// TwinCAT 3 PLC project Untitled1
// ProgramVersion: 3.1.4023.0
// libraries:
//   Tc2_Standard, * (Beckhoff Automation GmbH)
//   Tc2_System, * (Beckhoff Automation GmbH)
//   Tc3_Module, * (Beckhoff Automation GmbH)
//   VisuSymbols,3.5.10.0,System
// project tree:
//   / GlobalTextList.TcGTLO, PlcTask.TcTTO, RecipeManager.TcRMO (not stored), Visualization Manager.TcVMO (not stored), VISU_TASK.TcTTO
//   GVLs/ Recipes.TcGVL
//   POUs/ FB_PIZZA_OVEN.TcPOU, MAIN.TcPOU
//   VISUs/ OvenSimulation.TcVIS

CONFIGURATION Untitled1
    RESOURCE PLC ON TwinCAT3
        TASK PlcTask(INTERVAL := T#10ms, PRIORITY := 20);
        TASK VISU_TASK(INTERVAL := T#200000us, PRIORITY := 30);
        PROGRAM MAIN WITH PlcTask : MAIN;
        PROGRAM VisuElems_Visu_Prg WITH VISU_TASK : VisuElems.Visu_Prg;
    END_RESOURCE
END_CONFIGURATION

// ---- GVLs/Recipes.TcGVL
{attribute 'qualified_only'}
VAR_GLOBAL
END_VAR

// ---- POUs/MAIN.TcPOU
PROGRAM MAIN
VAR

	fbMyPizzaOven:FB_PIZZA_OVEN; //oven 1
	fbMyPizzaOven2:FB_PIZZA_OVEN; //oven 2
	btn_PutAPizza:BOOL;
	btn_PackageThePizza:BOOL;
	bReset:BOOL;
	
	btn_PutAPizzaT:R_TRIG;
	btn_PackageThePizzaT:R_TRIG;
	bResetT:R_TRIG;
	
	fbReadRecipe:RecipeManCommands;
	btnLoadRecipe:BOOL;
	btnSaveRecipe:BOOL;
	iIndexRecipe:int;
END_VAR

btn_PutAPizzaT(CLK:=main.btn_PutAPizza);
btn_PackageThePizzaT(CLK:=main.btn_PackageThePizza);
bResetT(CLK:=main.bReset);

fbMyPizzaOven(
	bReset:=main.bResetT.Q,
	btn_PutAPizza:=main.btn_PutAPizzaT.Q,
	btn_PackageThePizza:=main.btn_PackageThePizzaT.Q
);

fbMyPizzaOven2(
	bReset:=main.bResetT.Q,
	btn_PutAPizza:=main.btn_PutAPizzaT.Q,
	btn_PackageThePizza:=main.btn_PackageThePizzaT.Q
);

IF btnSaveRecipe THEN
	fbReadRecipe.ReadRecipe(
		RecipeDefinitionName:='Recipe',
		RecipeName:='MyRec'
	);
END_IF


IF btnLoadRecipe THEN
	fbReadRecipe.WriteRecipe(
		RecipeDefinitionName:='Recipe',
		RecipeName:='MyRec'
	);
END_IF

END_PROGRAM

// ---- POUs/FB_PIZZA_OVEN.TcPOU
 FUNCTION_BLOCK FB_PIZZA_OVEN

VAR_INPUT
	btn_PutAPizza:BOOL;
	btn_PackageThePizza:BOOL;
	bReset:BOOL;
	iFlavor:INT;
	iTime4Cooking:DINT:=1;
END_VAR


VAR_OUTPUT
		iTotalPizzasCooked :UDINT;
		iTotalPizzasBurned :UDINT;
		InpCookingTime:DINT;
		sCookingTime :DINT;
		LightCooking:BOOL;
 		LBuzzer:BOOL;
		sStateDescription :STRING;
		sPizzaDescription :STRING;
		sPizzaDescription2 :STRING;
END_VAR


VAR
	fbMyTimer : TON; //timer
	iState : DINT;
	bs_PizzaOnEntrit : BOOL;
	bs_PizzaOnOven : BOOL;
	bs_PizzaOnExit : BOOL;
	bBurnt :BOOL;
	bBurnt2 :BOOL;
	tTime4Cooking:TIME;
	bFlavor1:BOOL:=FALSE;
	bFlavor2:BOOL:=FALSE;
	bFlavor3:BOOL:=FALSE;
END_VAR

tTime4Cooking:=DINT_TO_TIME(iTime4Cooking*1000);

IF btn_PutAPizza THEN
	bs_PizzaOnEntrit:=TRUE;
	IF int_to_bool(iFlavor) THEN
		bFlavor1:=TRUE;
	ELSE
		bFlavor1:=FALSE;	
	END_IF
END_IF

IF btn_PackageThePizza THEN
	bs_PizzaOnExit:=FALSE;
	bFlavor3:=FALSE;
END_IF

IF bReset THEN
	bReset:=FALSE;
	iTotalPizzasCooked:=0;
	iTotalPizzasBurned:=0;
END_IF


CASE iState OF

	0: //wait for raw pizza 
		
		sStateDescription:='Waiting for pizza';
		IF bs_PizzaOnEntrit THEN
			IF bs_PizzaOnOven=FALSE THEN
				iState:=1;	
			END_IF
		END_IF
		
	1: //moving pizza
	
		sStateDescription:='Moving pizza';
		fbMyTimer(IN := TRUE,PT:=T#1S);
		IF fbMyTimer.Q THEN
			bs_PizzaOnOven:=TRUE;
			fbMyTimer(IN := FALSE);
			iState:=10;
			bs_PizzaOnEntrit:=FALSE;
			IF bFlavor1 THEN
				bFlavor2:=TRUE;
				bFlavor1:=FALSE;
			END_IF
		END_IF
		
	10: //there is a pizza, cook it
		
		sStateDescription:='Baking pizza';
		sPizzaDescription:='cooking';
		bBurnt:=false;
		LightCooking:=TRUE;
		sCookingTime:=(TIME_TO_DINT(fbMyTImer.ET))/1000;
		fbMyTimer(IN := TRUE,PT:=tTime4Cooking);
		IF fbMyTimer.Q THEN
			fbMyTimer(IN := FALSE);
			if bs_PizzaOnExit then
				iState:=20;
			else
				iState:=21;
			END_IF
			LightCooking:=FALSE;
			sCookingTime:=0;
		END_IF
		
	20: //burning pizza
	
		sStateDescription:='Pizza done, burning';
		sPizzaDescription:='burning';
		bBurnt:=true;
		IF NOT bs_PizzaOnExit THEN
			//simulating a conveyor
			bs_PizzaOnOven:=FALSE;
			bs_PizzaOnExit:=TRUE;
			IF bFlavor2 THEN
				bFlavor3:=TRUE;
				bFlavor2:=FALSE;
			END_IF
			iTotalPizzasBurned := iTotalPizzasBurned + 1;
			iState:=30;
			LBuzzer:=FALSE;
			sPizzaDescription2:='burned';
			bBurnt2:=TRUE;
		ELSE
			LBuzzer:=TRUE;
		END_IF
		
	21: //not burned pizza
	    sPizzaDescription2:='cooked';
		bBurnt2:=FALSE;
		iState:=30;
		bs_PizzaOnOven:=FALSE;
		bs_PizzaOnExit:=TRUE;
		IF bFlavor2 THEN
			bFlavor3:=TRUE;
			bFlavor2:=FALSE;
		END_IF
		iTotalPizzasCooked := iTotalPizzasCooked + 1;
		iState:=30;
		LBuzzer:=FALSE;
	
	30: //pizza just removed on output tray
	
		sStateDescription:='Please pack the pizza!';
		iState:=0; //wait for another pizza
		
END_CASE

END_FUNCTION_BLOCK

// ---- GlobalTextList.TcGTLO
TEXTLIST GlobalTextList
  330 = '%d'
  251 = '%s'
  80 = 'Burning'
  848 = 'Cooking'
  93 = 'Cooking time'
  637 = 'Cooking time '
  553 = 'Cooking time %d'
  817 = 'Cooking time %t'
  834 = 'Cooking time (seconds)'
  689 = 'Elapsed Time'
  143 = 'Elapsed Time %s'
  731 = 'Insert Pizza'
  435 = 'Käse'
  542 = 'Load Recipe'
  604 = 'New pizza ready'
  754 = 'NInsert Pizza'
  599 = 'package pizza'
  89 = 'Package the Pizza'
  915 = 'pizza'
  856 = 'Pizza # %d'
  275 = 'Pizza # %i'
  870 = 'Pizza %s'
  362 = 'pizza (done)'
  593 = 'pizza (on deck)'
  836 = 'Pizza cooking'
  123 = 'Pizza Cooking'
  935 = 'Pizza done'
  86 = 'Pizza Done'
  212 = 'Pizza raw'
  436 = 'Pizza Raw'
  163 = 'Pizzas burned: %d'
  468 = 'Pizzas cooked: %d'
  680 = 'Pizzas cooked: %s'
  651 = 'Put a Pizza'
  284 = 'Put a pizza'
  792 = 'Rea Pizza'
  734 = 'Recipe1'
  283 = 'Recipe2'
  695 = 'Recipe3'
  657 = 'Reset Counter'
  50 = 'Reset counter'
  253 = 'Reset CounterPizza'
  280 = 'Save Recipe'
  601 = 'Schinken'
  97 = 'Take Pizza out'
  459 = 'take the pizza'
  419 = 'test'
  214 = 'Timer %d'
  901 = 'Timer %s'
  265 = 'Timer %t'
END_TEXTLIST

// ---- VISUs/OvenSimulation.TcVIS
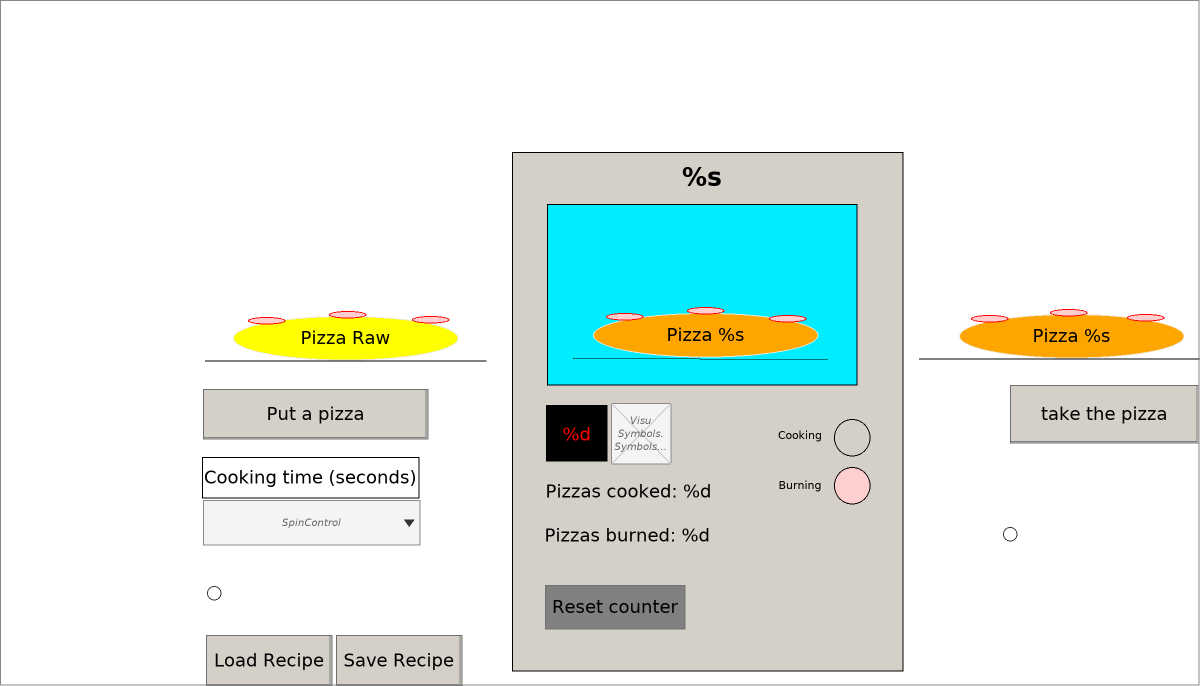
VISUALIZATION OvenSimulation  // 1200x686
    Rectangle (512,152 391x519)
    Ellipse (233,316 225x44), "Pizza Raw", invisible if: NOT main.fbMyPizzaOven.bs_PizzaOnEntrit
    Rectangle (546,405 61x56)
    Rectangle (547,204 310x181)
    Line (573,358) (827,359)
    Line (1200,359) (919,359)
    Line (486,361) (205,361)
    Ellipse (593,313 225x44), "Pizza %s", text variable: MAIN.fbMyPizzaOven.sPizzaDescription, colour toggle: MAIN.fbMyPizzaOven.bBurnt, invisible if: NOT main.fbMyPizzaOven.bs_PizzaOnOven
    Ellipse (834,419 36x37), colour toggle: MAIN.fbMyPizzaOven.LightCooking
    Ellipse (834,467 36x37), colour toggle: MAIN.fbMyPizzaOven.LBuzzer
    Label (744,403 112x65), "Cooking"
    Label (744,453 112x65), "Burning"
    Rectangle (497,413 160x43), "%d", text variable: MAIN.fbMyPizzaOven.sCookingTime, invisible if: not MAIN.fbMyPizzaOven.LightCooking
    Rectangle (507,153 390x47), "%s", text variable: MAIN.fbMyPizzaOven.sStateDescription
    Rectangle (517,468 223x47), "Pizzas cooked: %d", text variable: MAIN.fbMyPizzaOven.iTotalPizzasCooked
    Button (203,389 225x50), "Put a pizza"
        OnMouseDown: execute { main.btn_PutAPizza:=TRUE; }
        OnMouseUp: execute { main.btn_PutAPizza:=FALSE; }
    Button (1010,385 189x58), "take the pizza"
        OnMouseDown: execute { main.btn_PackageThePizza:=TRUE; }
        OnMouseUp: execute { main.btn_PackageThePizza:=FALSE; }
    Button (545,585 140x44), "Reset counter"
        OnMouseDown: execute { main.bReset:=TRUE; }
        OnMouseUp: execute { main.bReset:=FALSE; }
    Ellipse (959,314 225x44), "Pizza %s", text variable: MAIN.fbMyPizzaOven.sPizzaDescription2, colour toggle: MAIN.fbMyPizzaOven.bBurnt2, invisible if: NOT main.fbMyPizzaOven.bs_PizzaOnExit
    Rectangle (516,512 223x47), "Pizzas burned: %d", text variable: MAIN.fbMyPizzaOven.iTotalPizzasBurned
    Image (611,403 60x61), image: VisuSymbols.Symbols.Timer
    SpinControl (203,500 217x45), variable: MAIN.fbMyPizzaOven.iTime4Cooking
        p1653691745: .5
    Rectangle (202,457 217x41), "Cooking time (seconds)", text variable: MAIN.fbMyPizzaOven.tTime4Cooking
    RadioButton (205,557 196x72), variable: MAIN.fbMyPizzaOven.iFlavor
        Areas[0]: Text=Käse
        Areas[1]: Text=Schinken
    Ellipse (248,317 37x7), angle 349, invisible if: not MAIN.fbMyPizzaOven.bFlavor1
    Ellipse (329,311 37x7), invisible if: not MAIN.fbMyPizzaOven.bFlavor1
    Ellipse (412,316 37x7), angle 11, invisible if: not MAIN.fbMyPizzaOven.bFlavor1
    Ellipse (606,313 37x7), angle 349, invisible if: not MAIN.fbMyPizzaOven.bFlavor2
    Ellipse (769,315 37x7), angle 11, invisible if: not MAIN.fbMyPizzaOven.bFlavor2
    Ellipse (687,307 37x7), invisible if: not MAIN.fbMyPizzaOven.bFlavor2
    Ellipse (1050,309 37x7), invisible if: not MAIN.fbMyPizzaOven.bFlavor3
    Ellipse (1127,314 37x7), angle 11, invisible if: not MAIN.fbMyPizzaOven.bFlavor3
    Ellipse (971,315 37x7), angle 349, invisible if: not MAIN.fbMyPizzaOven.bFlavor3
    Button (206,635 126x51), "Load Recipe"
        tap MAIN.btnLoadRecipe
    Button (336,635 126x51), "Save Recipe"
        tap MAIN.btnSaveRecipe
    RadioButton (1001,485 158x98), variable: MAIN.iIndexRecipe
        Areas[0]: Text=Recipe1
        Areas[1]: Text=Recipe2
        Areas[2]: Text=Recipe3
END_VISUALIZATION
